{attribute addProperty BoxType "EL6201-0000-0017"}
{attribute addProperty Id "Slave_11A_DI0BIT10.12581Slave_11A_DI1BIT10.12582Slave_11A_DI2BIT10.12583Slave_11A_DI3BIT10.12584Slave_11B_DI0BIT10.12585Slave_11B_DI1BIT10.12586Slave_11B_DI2BIT10.12587Slave_11B_DI3BIT10.12588"}
{attribute addProperty CRC "3765272816"}
{attribute addProperty SizeInBites "8"}
{attribute addProperty SizeInBytes "1"}
TYPE Slave_11_Inputs_E06D80F0 :
STRUCT
	{attribute addProperty Name "Slave_11A_DI0"}
	Slave_11A_DI0 : BIT;
	{attribute addProperty Name "Slave_11A_DI1"}
	Slave_11A_DI1 : BIT;
	{attribute addProperty Name "Slave_11A_DI2"}
	Slave_11A_DI2 : BIT;
	{attribute addProperty Name "Slave_11A_DI3"}
	Slave_11A_DI3 : BIT;
	{attribute addProperty Name "Slave_11B_DI0"}
	Slave_11B_DI0 : BIT;
	{attribute addProperty Name "Slave_11B_DI1"}
	Slave_11B_DI1 : BIT;
	{attribute addProperty Name "Slave_11B_DI2"}
	Slave_11B_DI2 : BIT;
	{attribute addProperty Name "Slave_11B_DI3"}
	Slave_11B_DI3 : BIT;
END_STRUCT
END_TYPE

(* stored: Version 1.2.0.0, ProductVersion 3.1.4024.9
   DUT Slave_11_Inputs_E06D80F0: Id {5eaa67e4-5124-4368-be97-1651849feb00} *)
